// TIA Portal V15.1 export
// export: Created 2020-06-12T07:35:45.4599609Z, ExportSetting None, DisplayName Totally Integrated Automation Portal, DisplayVersion V15.1, DisplayName TIA Portal Openness, DisplayVersion V15.1, DisplayName STEP 7 Professional, DisplayVersion V15.1, DisplayName STEP 7 Safety, DisplayVersion V15.1, DisplayName WinCC Advanced, DisplayVersion V15.1
FUNCTION "Alloy_common" : Void   // FC160, FBD
{ S7_Optimized_Access := 'TRUE' }
// stored: SetENOAutomatically False
   VAR_TEMP
      tPwrOK : Bool;   // Emergency OK
      tRdyM01 : Bool;   // ES1LA2_M01 - Motor in Auto mode and no error
      tRdyM02 : Bool;   // ES1LA2_M02 - Motor in Auto mode and no error
      tRdyM03 : Bool;   // ES1LA2_M03 - Motor in Auto mode and no error
      tRdyEV01 : Bool;   // ES1LA2_EV01 - Valve in auto mode and no error
      tRdyEV02 : Bool;   // ES1LA2_EV02 - Valve in auto mode and no error
      tRdyEV03 : Bool;   // ES1LA2_EV03 - Valve in auto mode and no error
      tRdyEV08 : Bool;   // ES1LG1_EV08 - Valve in auto mode and no error
      _low : Real;
   END_VAR
   VAR_TEMP   // added for the SCL form of the ladder/FBD networks
      _w1 : Bool;
      _w2 : Bool;
   END_VAR
BEGIN

REGION Network 2: Power supply
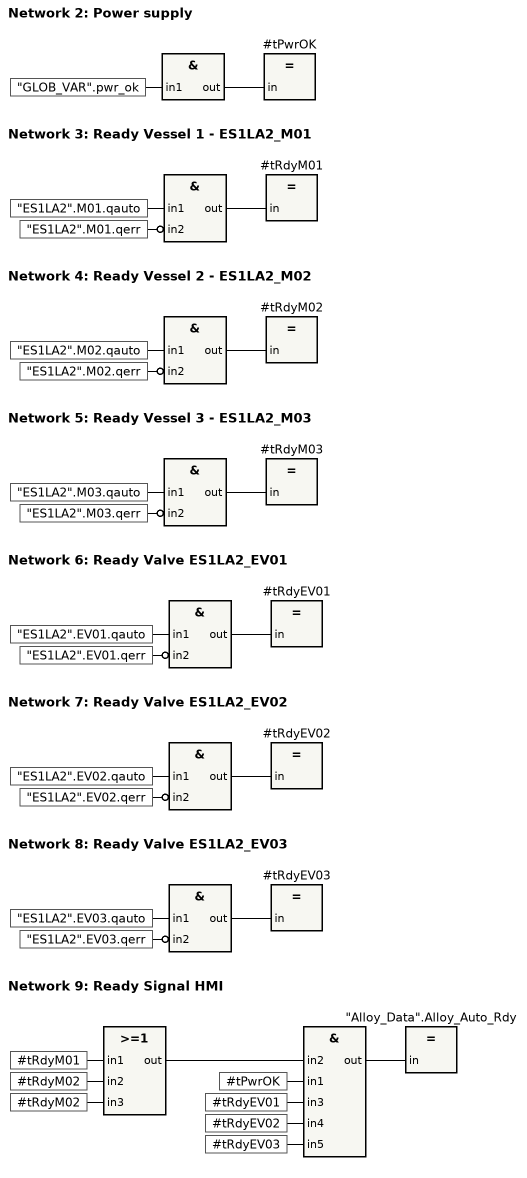
   #tPwrOK := "GLOB_VAR".pwr_ok;
END_REGION

REGION Network 3: Ready Vessel 1 - ES1LA2_M01
   #tRdyM01 := "ES1LA2".M01.qauto AND NOT "ES1LA2".M01.qerr;
END_REGION

REGION Network 4: Ready Vessel 2 - ES1LA2_M02
   #tRdyM02 := "ES1LA2".M02.qauto AND NOT "ES1LA2".M02.qerr;
END_REGION

REGION Network 5: Ready Vessel 3 - ES1LA2_M03
   #tRdyM03 := "ES1LA2".M03.qauto AND NOT "ES1LA2".M03.qerr;
END_REGION

REGION Network 6: Ready Valve ES1LA2_EV01
   #tRdyEV01 := "ES1LA2".EV01.qauto AND NOT "ES1LA2".EV01.qerr;
END_REGION

REGION Network 7: Ready Valve ES1LA2_EV02
   #tRdyEV02 := "ES1LA2".EV02.qauto AND NOT "ES1LA2".EV02.qerr;
END_REGION

REGION Network 8: Ready Valve ES1LA2_EV03
   #tRdyEV03 := "ES1LA2".EV03.qauto AND NOT "ES1LA2".EV03.qerr;
END_REGION

REGION Network 9: Ready Signal HMI
   "Alloy_Data".Alloy_Auto_Rdy := (#tRdyM01 OR #tRdyM02 OR #tRdyM02) AND #tPwrOK AND #tRdyEV01 AND #tRdyEV02 AND #tRdyEV03;
END_REGION

REGION Network 10: Alloy auto ON in Premelt
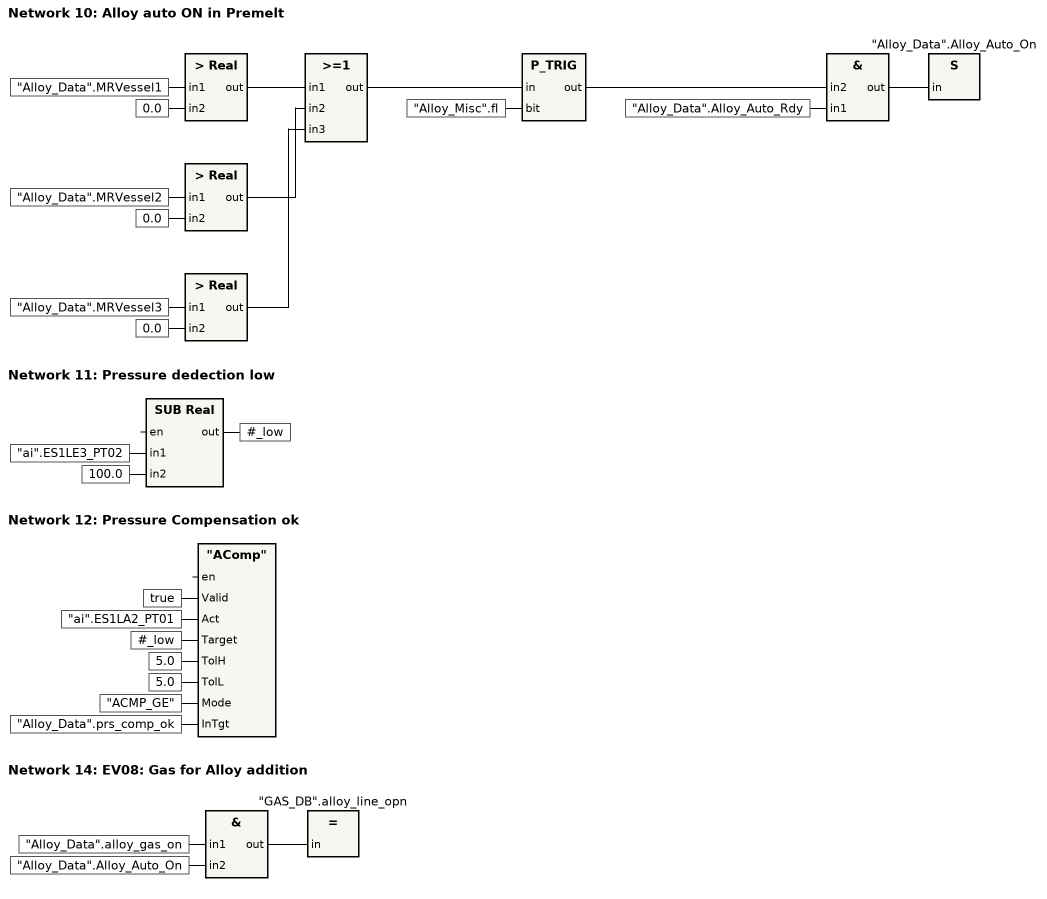
   #_w1 := ("Alloy_Data".MRVessel1 > 0.0) OR ("Alloy_Data".MRVessel2 > 0.0) OR ("Alloy_Data".MRVessel3 > 0.0);
   #_w2 := #_w1 AND NOT "Alloy_Misc".fl;   // rising edge
   "Alloy_Misc".fl := #_w1;
   IF #_w2 AND "Alloy_Data".Alloy_Auto_Rdy THEN "Alloy_Data".Alloy_Auto_On := TRUE; END_IF;
END_REGION

REGION Network 11: Pressure dedection low
   #_low := "ai".ES1LE3_PT02 - 100.0;
END_REGION

REGION Network 12: Pressure Compensation ok
   "AComp"(Valid := true,
           Act := "ai".ES1LA2_PT01,
           Target := #_low,
           TolH := 5.0,
           TolL := 5.0,
           Mode := "ACMP_GE",
           InTgt := "Alloy_Data".prs_comp_ok);
END_REGION

REGION Network 13: Calculate g per Cycle from Meltrate
END_REGION

REGION Network 14: EV08: Gas for Alloy addition
   "GAS_DB".alloy_line_opn := "Alloy_Data".alloy_gas_on AND "Alloy_Data".Alloy_Auto_On;
END_REGION
END_FUNCTION
